FUNCTION_BLOCK logiBUS_IE2A (* Composite FB for event input data with argument *)
  (* Standard: 61499-2; Description: Copyright (c) 2026 HR Agrartechnik GmbH This program and the accompanying materials are made available under the terms of the Eclipse Public License 2.0 which is available at https://www.eclipse.org/legal/epl-2.0/ SPDX-License-Identifier: EPL-2.0 *)
  (* Version 1.0, 2026-02-23, Franz Höpfinger, HR Agrartechnik GmbH *)
  PACKAGE logiBUS::io::DI;
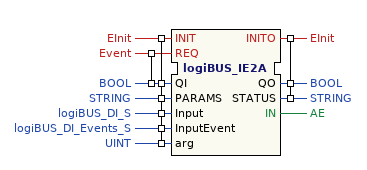
  EVENT_INPUT
    INIT : EInit WITH QI, PARAMS, Input, InputEvent, arg; (* Service Initialization *)
    REQ WITH QI; (* Service Request *)
  END_EVENT
  EVENT_OUTPUT
    INITO : EInit WITH QO, STATUS; (* Initialization Confirm *)
  END_EVENT
  VAR_INPUT
    QI : BOOL; (* Event Input Qualifier *)
    PARAMS : STRING; (* Service Parameters *)
    Input : logiBUS::io::DI::logiBUS_DI_S := logiBUS_DI::Invalid; (* Identify the Input Input_I1..I8 *)
    InputEvent : logiBUS::io::DI::logiBUS_DI_Events_S := logiBUS_DI_Events::Invalid; (* Identify the Event (Down, Up, Single-Click, Double Click etc..) *)
    arg : UINT := 65535; (* Long press time event data OR Multiple clicks event data (Depending on Input Event) *)
  END_VAR
  VAR_OUTPUT
    QO : BOOL; (* Event Output Qualifier *)
    STATUS : STRING; (* Service Status *)
  END_VAR
  PLUGS
    IN : adapter::types::unidirectional::AE;
  END_PLUGS
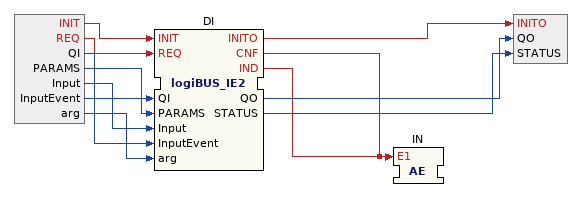
  FBS
    DI : logiBUS::io::DI::logiBUS_IE2;
  END_FBS
  EVENT_CONNECTIONS
    INIT TO DI.INIT;
    DI.INITO TO INITO;
    DI.IND TO IN.E1;
    DI.CNF TO IN.E1;
    REQ TO DI.REQ;
  END_CONNECTIONS
  DATA_CONNECTIONS
    QI TO DI.QI;
    PARAMS TO DI.PARAMS;
    DI.QO TO QO;
    DI.STATUS TO STATUS;
    Input TO DI.Input;
    InputEvent TO DI.InputEvent;
    arg TO DI.arg;
  END_CONNECTIONS
END_FUNCTION_BLOCK
